(* CoDeSys 2.3 export: PODPITKA.EXP *)

(* POU Podpitka, ST *)
PROGRAM Podpitka
VAR
END_VAR

END_PROGRAM
